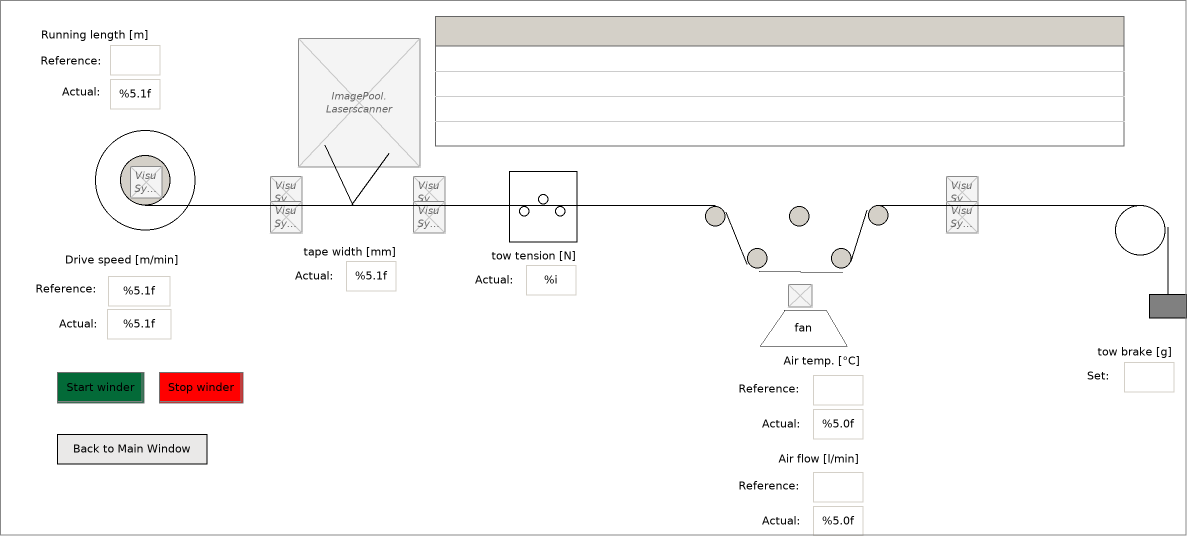
VISUALIZATION Setup_Mode  // 1187x536
    Label (20,20 150x30), "Running length [m]"
    Textfield (110,45 50x30)
    Label (47,245 150x30), "Drive speed [m/min]"
    Textfield (107,309 64x30), "%5.1f", text variable: GVL_HMI.ActTapeSpeed
        OnMouseClick: write the text variable via Default
    Label (24,46 80x30), "Reference:"
    Label (23,77 80x30), "Actual:"
    Ellipse (95,130 100x100)
    Ellipse (120,155 50x50)
    Label (20,309 80x30), "Actual:"
    Label (19,274 80x30), "Reference:"
    Image (270,176 32x32), image: VisuSymbols.Symbols.TriangleDown
    Image (270,201 32x32), image: VisuSymbols.Symbols.TriangleUp
    Image (413,176 32x32), image: VisuSymbols.Symbols.TriangleDown
    Image (413,201 32x32), image: VisuSymbols.Symbols.TriangleUp
    Ellipse (705,206 20x20)
    Ellipse (747,248 20x20)
    Ellipse (789,206 20x20)
    Ellipse (831,248 20x20)
    Ellipse (868,205 20x20)
    Image (946,176 32x32), image: VisuSymbols.Symbols.TriangleDown
    Image (946,201 32x32), image: VisuSymbols.Symbols.TriangleUp
    Label (763,346 100x30), "Air temp. [°C]"
    Textfield (813,409 50x30), "%5.0f", text variable: GVL_Axis.rWinderVelocity
        OnMouseClick: write the text variable via Default
    Textfield (813,375 50x30)
    Label (723,409 80x30), "Actual:"
    Label (722,374 80x30), "Reference:"
    Label (762,444 100x30), "Air flow [l/min]"
    Textfield (813,506 50x30), "%5.0f", text variable: GVL_Axis.rWinderVelocity
        OnMouseClick: write the text variable via Default
    Textfield (813,472 50x30)
    Label (723,506 80x30), "Actual:"
    Label (722,471 80x30), "Reference:"
    Label (285,237 114x30), "tape width [mm]"
    Textfield (346,261 50x30), "%5.1f", text variable: GVL_Axis.rWinderVelocity
        OnMouseClick: write the text variable via Default
    Label (256,261 80x30), "Actual:"
    Polygon (785,310) (784,310) (826,310) (847,346) (760,346), "fan"
    Image (788,284 24x23), image: VisuSymbols.Symbols.ArrowBoldUp
    Line (747,264) (726,212)
    Line (759,271) (842,272)
    Label (465,241 114x30), "tow tension [N]"
    Textfield (526,265 50x30), "%i", text variable: GVL.iTensionMonitoringData
        OnMouseClick: write the text variable via Default
    Label (436,265 80x30), "Actual:"
    Label (1061,337 114x30), "tow brake [g]"
    Label (1032,361 80x30), "Set:"
    Textfield (1124,362 50x30)
    Table (435,16 689x130), data array: GVL.LaserScannerData
        p3854506369: GVL.LaserScannerData[INDEX]
    Rectangle (57,434 150x30), "Back to Main Window"
        OnMouseClick: change screen: MainWindow
    Textfield (110,79 50x30), "%5.1f", text variable: GVL_HMI.RunningLength
        OnMouseClick: write the text variable via Default
    Rectangle (509,171 68x71)
    Ellipse (519,206 10x10)
    Ellipse (538,194 10x10)
    Ellipse (555,206 10x10)
    Line (145,205) (715,205)
    Line (851,261) (867,210)
    Line (877,205) (1142,205)
    Ellipse (1115,205 50x50)
    Line (1168,298) (1168,227)
    Rectangle (1149,294 38x24)
    Image (298,38 122x129), image: ImagePool.Laserscanner
    Line (352,204) (389,153)
    Line (353,205) (325,145)
    Textfield (108,276 62x30), "%5.1f", text variable: GVL_Axis.rWinderVelocity
        OnMouseClick: write the text variable via VisuDialogs.Numpad, min 2.7, max 15
    Button (57,372 87x31), "Start winder", colour toggle: GVL_HMI.bButtonStartWinder
        OnMouseDown: execute { GVL_HMI.bButtonStartWinder := TRUE; }
        OnMouseUp: execute { GVL_HMI.bButtonStartWinder := FALSE; }
    Button (159,372 84x31), "Stop winder", colour toggle: GVL_HMI.bButtonStopWinder
        OnMouseDown: execute { GVL_HMI.bButtonStopWinder := TRUE; }
        OnMouseUp: execute { GVL_HMI.bButtonStopWinder := FALSE; }
    Image (130,166 32x32), image: VisuSymbols.Symbols.ArrowHalfRightUp
END_VISUALIZATION

(* stored: Version 1.1.0.1
   Visu Setup_Mode: Id {7f124c42-37b8-4992-b74a-a9c898da625d} *)
